INTERFACE IController EXTENDS IOut

METHOD Update : IOut
VAR_INPUT
    setpoint : LREAL;
    actual : LREAL;
END_VAR
END_METHOD

END_INTERFACE

(* stored: Version 1.1.0.1, ProductVersion 3.1.4024.12
   Itf IController: Id {6d4eca49-a523-4b77-8ac2-546b7813c75c}
   Method Update: Id {98645dea-5ead-4697-a969-ccba5550c9ef} *)
